(* IEC 61131-3 sources: automationbase/test/mocks, 8 files *)

(* ---- TimestampMock.st ---- *)
USING System.DateTime;

NAMESPACE Simatic.Ax.Mocks

    /// Mock for GetCurrentTimestamp that returns a fixed timestamp
    FUNCTION GetCurrentTimestamp : LDATE_AND_TIME
        // Return a fixed timestamp for testing: 2024-01-15 10:30:45
        GetCurrentTimestamp := LDATE_AND_TIME#2024-01-15-10:30:45;
    END_FUNCTION

END_NAMESPACE

(* ---- MockingAutoRelease.st ---- *)
NAMESPACE Simatic.Ax.AutomationBase

    CLASS MockAutoReleaseIsReleased
        IMPLEMENTS IRelease

        METHOD PUBLIC IsReleased : BOOL
            IsReleased := TRUE;;
        END_METHOD
    END_CLASS
END_NAMESPACE

(* ---- MockingAutoStartup.st ---- *)
USING Simatic.Ax.AutomationBase;

NAMESPACE Simatic.Ax.Conveyor.Mocks

    /// <summary>
    /// Mock implementation of IAutoStartup interface for testing.
    /// Allows tests to control the startup status returned by the Status() method.
    /// </summary>
    CLASS MockAutoStartup
        IMPLEMENTS IAutoStartup
        VAR PUBLIC
            /// Configurable startup status that will be returned by Status() method
            startupStatus : StartUpStatus := StartUpStatus#NotReleased;
        END_VAR

        /// <summary>
        /// Returns the configured startup status.
        /// </summary>
        /// <returns>The current value of startupStatus</returns>
        METHOD PUBLIC Status : StartUpStatus
            Status := startupStatus;
        END_METHOD
    END_CLASS

END_NAMESPACE

(* ---- MockingEquipment.st ---- *)
USING Simatic.Ax.AutomationBase;
NAMESPACE Simatic.Ax.Conveyor.Mocks

    CLASS MockEquiment
        IMPLEMENTS IEquipmentBase
        VAR PUBLIC
            MockError : BOOL;
            MockStatus : StartUpStatus;
        END_VAR
        VAR PROTECTED
            _error : BOOL;
            _errorText : STRING[30];
        END_VAR

        METHOD PUBLIC HasError : BOOL
            HasError := MockError;
        END_METHOD

        METHOD PUBLIC GetStartupStatus : StartUpStatus
            GetStartupStatus := MockStatus;
        END_METHOD

        METHOD PUBLIC GetError : ErrorState
            ;
        END_METHOD

        METHOD PUBLIC GetErrorText : STRING[30]
            GetErrorText := _errorText;
        END_METHOD

        METHOD PUBLIC Init
            ;
        END_METHOD

        METHOD PUBLIC RunCyclic
            ;
        END_METHOD

        METHOD PUBLIC ResetFault
            _error := FALSE;
            _errorText := '';
        END_METHOD

        METHOD PUBLIC SetError
            VAR_INPUT
                errorState : ErrorState;
            END_VAR
            _error := TRUE;
            _errorText := '';
        END_METHOD

        METHOD PUBLIC SetError
            VAR_INPUT
                errorState : ErrorState;
                errorText : STRING[30];
            END_VAR
            _error := TRUE;
            _errorText := errorText;
        END_METHOD
    END_CLASS

END_NAMESPACE

(* ---- MockingEquipmentBase.st ---- *)
USING Simatic.Ax.AutomationBase;
NAMESPACE Simatic.Ax.Conveyor.Mocks

    /// <summary>
    /// Concrete implementation of the abstract EquipmentBase class for testing purposes.
    /// This mock tracks method calls and provides counters for test verification.
    /// </summary>
    CLASS MockEquipmentBase EXTENDS EquipmentBase
        VAR PUBLIC
            /// Flag indicating if RunCyclicUserCode was called at least once
            RunCyclicUserCodeCalled : BOOL;
            /// Flag indicating if InitUser was called at least once
            InitUserCalled : BOOL;
            /// Counter tracking how many times RunCyclicUserCode was called
            RunCyclicUserCodeCallCount : INT;
            /// Counter tracking how many times InitUser was called
            InitUserCallCount : INT;
        END_VAR

        /// <summary>
        /// Override of the abstract RunCyclicUserCode method.
        /// Sets the called flag and increments the call counter for test verification.
        /// </summary>
        METHOD PROTECTED OVERRIDE RunCyclicUserCode
            RunCyclicUserCodeCalled := TRUE;
            RunCyclicUserCodeCallCount := RunCyclicUserCodeCallCount + 1;
        END_METHOD

        /// <summary>
        /// Override of the abstract InitUser method.
        /// Sets the called flag and increments the call counter for test verification.
        /// </summary>
        METHOD PROTECTED OVERRIDE InitUser
            InitUserCalled := TRUE;
            InitUserCallCount := InitUserCallCount + 1;
        END_METHOD

        /// <summary>
        /// Helper method to reset all test tracking flags and counters.
        /// Should be called in test setup to ensure clean state between tests.
        /// </summary>
        METHOD PUBLIC ResetTestFlags
            RunCyclicUserCodeCalled := FALSE;
            InitUserCalled := FALSE;
            RunCyclicUserCodeCallCount := 0;
            InitUserCallCount := 0;
        END_METHOD

        METHOD PROTECTED OVERRIDE ResetFaultUser : BOOL
            ResetFaultUser := TRUE;
        END_METHOD
    END_CLASS

END_NAMESPACE

(* ---- MockingOperatingModes.st ---- *)
USING Simatic.Ax.AutomationBase;
NAMESPACE Simatic.Ax.Conveyor.Mocks

    CLASS MockOperatingMode
        IMPLEMENTS IOperatingMode
        VAR PUBLIC
            mode : OperatingModes;
        END_VAR
        METHOD PUBLIC GetOperatingMode : OperatingModes
            GetOperatingMode := mode;
        END_METHOD
    END_CLASS
END_NAMESPACE

(* ---- MockingRelese.st ---- *)
USING Simatic.Ax.AutomationBase;
NAMESPACE Simatic.Ax.Conveyor.Mocks

    CLASS MockIsReleased_TRUE
        IMPLEMENTS IRelease
        METHOD PUBLIC IsReleased : BOOL
            IsReleased := TRUE;
        END_METHOD
    END_CLASS
    CLASS MockIsReleased_FALSE
        IMPLEMENTS IRelease
        METHOD PUBLIC IsReleased : BOOL
            IsReleased := FALSE;
        END_METHOD
    END_CLASS

END_NAMESPACE

(* ---- OnDelayMock_passthrough.st ---- *)
NAMESPACE Simatic.Ax.Mocks
    /// Mock für OnDelay Timer - verhält sich wie echter Timer
    /// Gibt TRUE zurück wenn signal TRUE ist
    FUNCTION_BLOCK OnDelayMock_passthrough
        VAR_INPUT
            duration : LTIME;
            signal : BOOL;
        END_VAR
        VAR_OUTPUT
            output : BOOL;
            elapsedTime : LTIME;
        END_VAR
        output := signal;
    END_FUNCTION_BLOCK
END_NAMESPACE
